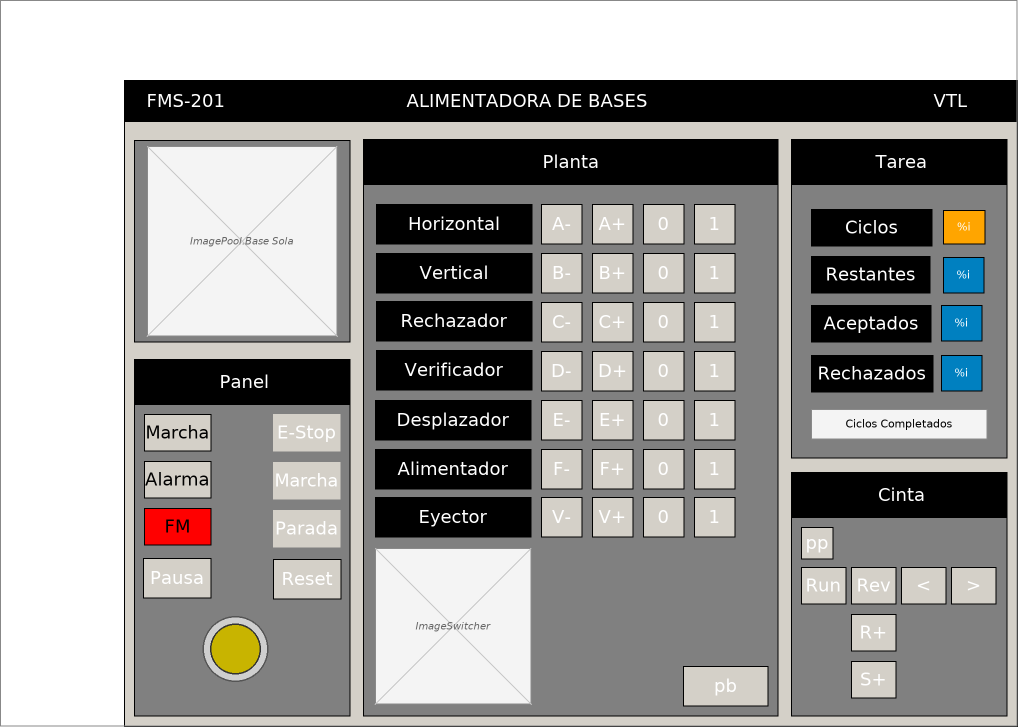
VISUALIZATION Visualization  // 1018x727
    Rectangle (124,121 894x606)
    Rectangle (791,184 216x274)
    Rectangle (363,184 415x532)
    Rectangle (363,139 415x45)
    Label (363,141 416x42), "Planta"
    Rectangle (791,139 216x45)
    Label (841,144 121x36), "Tarea"
    Progressbar (811,409 176x30), "Ciclos Completados", variable: MAIN.test_pieza.Aceptados
    RoundedRectangle (376,204 156x40), "Horizontal"
    Textfield (943,210 42x34), "%i", text variable: MAIN.Estacion.CiclosSolicitados
        OnMouseDown: write MAIN.Estacion.CiclosSolicitados via VisuDialogs.Numpad, min 1, max 10
    RoundedRectangle (811,209 121x37), "Ciclos"
    RoundedRectangle (811,256 119x37), "Restantes"
    RoundedRectangle (811,305 120x37), "Aceptados"
    RoundedRectangle (811,355 122x37), "Rechazados"
    Textfield (943,257 41x36), "%i", text variable: MAIN.Estacion.CiclosPendientes
    Textfield (941,305 41x36), "%i", text variable: MAIN.Estacion.CiclosAceptados
    Textfield (941,355 41x36), "%i", text variable: MAIN.Estacion.CiclosRechazados
    RoundedRectangle (592,253 41x40), "B+", colour toggle: MAIN.Estacion.Descargador_baja
        toggle MAIN.Estacion.Descargador_baja
    Rectangle (791,517 216x199)
    Rectangle (791,472 216x45)
    Label (841,477 121x36), "Cinta"
    Rectangle (134,140 216x202)
    Rectangle (134,404 216x312)
    Rectangle (134,359 216x45)
    Label (184,364 121x36), "Panel"
    Rectangle (124,80 894x41)
    Label (124,81 893x40), "FMS-201 ALIMENTADORA DE BASES VTL"
    RoundedRectangle (376,253 156x40), "Vertical"
    RoundedRectangle (592,204 41x40), "A+", colour toggle: MAIN.Estacion.Descargador_adelante
        tap MAIN.Estacion.Descargador_adelante
    RoundedRectangle (592,302 41x40), "C+", colour toggle: MAIN.Estacion.Rechazador_adelante
        tap MAIN.Estacion.Rechazador_adelante
    RoundedRectangle (592,351 41x40), "D+", colour toggle: MAIN.Estacion.Verificador_baja
        tap MAIN.Estacion.Verificador_baja
    RoundedRectangle (592,400 41x40), "E+", colour toggle: MAIN.Estacion.Desplazador_adelante
        tap MAIN.Estacion.Desplazador_adelante
    RoundedRectangle (592,449 41x40), "F+", colour toggle: MAIN.Estacion.Alimentador_adelante
        tap MAIN.Estacion.Alimentador_adelante
    RoundedRectangle (592,497 41x40), "V+", colour toggle: MAIN.Estacion.Eyector_succiona
        toggle MAIN.Estacion.Eyector_succiona
    RoundedRectangle (376,301 156x40), "Rechazador"
    RoundedRectangle (376,350 156x40), "Verificador"
    RoundedRectangle (375,400 156x40), "Desplazador"
    RoundedRectangle (375,449 156x40), "Alimentador"
    RoundedRectangle (375,497 156x40), "Eyector"
    RoundedRectangle (541,204 41x40), "A-", colour toggle: MAIN.Estacion.Descargador_atras
        tap MAIN.Estacion.Descargador_atras
    RoundedRectangle (643,204 41x40), "0", colour toggle: MAIN.Estacion.Horizontal_descargador_detras
    RoundedRectangle (694,204 41x40), "1", colour toggle: MAIN.Estacion.Horizontal_descargador_delante
    RoundedRectangle (643,253 41x40), "0", colour toggle: MAIN.Estacion.Vertical_descargador_arriba
        tap MAIN.Estacion.Vertical_descargador_arriba
    RoundedRectangle (694,253 41x40), "1", colour toggle: MAIN.Estacion.Vertical_descargador_abajo
        tap MAIN.Estacion.Vertical_descargador_abajo
    RoundedRectangle (643,302 41x40), "0"
    RoundedRectangle (643,351 41x40), "0", colour toggle: MAIN.Estacion.Verificador_arriba
        tap MAIN.Estacion.Verificador_arriba
    RoundedRectangle (643,400 41x40), "0", colour toggle: MAIN.Estacion.Desplazador_detras
        tap MAIN.Estacion.Desplazador_detras
    RoundedRectangle (643,449 41x40), "0", colour toggle: MAIN.Estacion.Alimentador_detras
        tap MAIN.Estacion.Alimentador_detras
    RoundedRectangle (643,497 41x40), "0"
    RoundedRectangle (694,302 41x40), "1"
    RoundedRectangle (694,351 41x40), "1", colour toggle: MAIN.Estacion.Verificador_abajo
        tap MAIN.Estacion.Verificador_abajo
    RoundedRectangle (694,400 41x40), "1"
    RoundedRectangle (694,449 41x40), "1", colour toggle: MAIN.Estacion.Alimentador_delante
        tap MAIN.Estacion.Alimentador_delante
    RoundedRectangle (694,497 41x40), "1", colour toggle: MAIN.Estacion.Vacio_obtenido_vacuostato_descargador
        tap MAIN.Estacion.Vacio_obtenido_vacuostato_descargador
    RoundedRectangle (541,253 41x40), "B-"
    RoundedRectangle (541,302 41x40), "C-"
    RoundedRectangle (541,351 41x40), "D-"
    RoundedRectangle (541,400 41x40), "E-"
    RoundedRectangle (541,449 41x40), "F-"
    RoundedRectangle (541,497 41x40), "V-"
    RoundedRectangle (683,666 85x40), "pb", colour toggle: MAIN.Estacion.Base_en_Alimentador
        tap MAIN.Estacion.Base_en_Alimentador
    RoundedRectangle (144,508 67x37), "FM", colour toggle: MAIN.Estacion.Lampara_falta_material
        tap MAIN.Estacion.Lampara_falta_material
    RoundedRectangle (801,527 32x32), "pp", colour toggle: MAIN.Estacion.Presencia_pale
        tap MAIN.Estacion.Presencia_pale
    RoundedRectangle (951,567 45x37), ">", colour toggle: MAIN.Estacion.Activa_marcha_motor_cinta
        tap MAIN.Estacion.Activa_marcha_motor_cinta
    RoundedRectangle (901,567 45x37), "<", colour toggle: MAIN.Estacion.Invierte_marcha_motor_cinta
        toggle MAIN.Estacion.Invierte_marcha_motor_cinta
    RoundedRectangle (801,567 45x37), "Run", colour toggle: MAIN.Estacion.Activa_marcha_motor_cinta
    RoundedRectangle (851,567 45x37), "Rev", colour toggle: MAIN.Estacion.Invierte_marcha_motor_cinta
    RoundedRectangle (851,614 45x37), "R+", colour toggle: MAIN.Estacion.Retenedor_pale_baja
        toggle MAIN.Estacion.Retenedor_pale_baja
    RoundedRectangle (851,661 45x37), "S+", colour toggle: MAIN.Estacion.Separador_pale_sube
        toggle MAIN.Estacion.Separador_pale_sube
    RoundedRectangle (273,414 67x37), "E-Stop", colour toggle: MAIN.Estacion.Pulsador_parada_emergencia
        tap MAIN.Estacion.Pulsador_parada_emergencia
    RoundedRectangle (273,462 67x37), "Marcha", colour toggle: MAIN.Estacion.Pulsador_marcha
        tap MAIN.Estacion.Pulsador_marcha
    RoundedRectangle (273,510 67x37), "Parada", colour toggle: MAIN.Estacion.Pulsador_parada_NC
        tap MAIN.Estacion.Pulsador_parada_NC
    RoundedRectangle (144,461 67x37), "Alarma", colour toggle: MAIN.Estacion.Lampara_alarma
        tap MAIN.Estacion.Lampara_alarma
    RoundedRectangle (144,414 67x37), "Marcha", colour toggle: MAIN.Estacion.Lampara_marcha
        tap MAIN.Estacion.Lampara_marcha
    Image (147,146 190x190), image: ImagePool.Base Sola
    Lamp1 (197,611 77x76), variable: MAIN.test_pieza.Lampara_falta_material, style: Lamp-Lamp1-Yellow
    ImageSwitcher (375,548 156x156), variable: MAIN.Estacion.pieza_ok, background image: ImagePool.Base OK, image: ImagePool.Base No OK, behaviour: TOGGLE
    RoundedRectangle (143,558 68x40), "Pausa", text variable: MAIN.Estacion.EstadoPausa, colour toggle: MAIN.Estacion.EstadoPausaMAIN.Estacion.EstadoPausa
        tap MAIN.Estacion.EstadoPausa
    RoundedRectangle (273,559 68x40), "Reset", text variable: MAIN.Estacion.EstadoReinicia, colour toggle: MAIN.Estacion.EstadoReinicia
        tap MAIN.Estacion.EstadoReinicia
END_VISUALIZATION

(* stored: Version 1.1.0.1, ProductVersion 3.1.4024.12
   Visu Visualization: Id {58b9ed46-5411-481b-9635-3712a23a6673} *)
